TYPE ST_Zustand_Netz_Anford :
STRUCT
	Aktiv				: BOOL	;
	Temp                : REAL;
	Temp_Max            : REAL;
	Temp_Min            : REAL;
	Temp_Oben			: REAL;
	Temp_Oben_Max		: REAL	;
	Temp_Oben_Min		: REAL	;
	Temp_Unten			: REAL;
	Temp_Unten_Max		: REAL	;
	Temp_Unten_Min		: REAL	;
END_STRUCT
END_TYPE

(* stored: Version 1.1.0.1, ProductVersion 3.1.4024.10
   DUT ST_Zustand_Netz_Anford: Id {3bb66fe0-892b-4f8e-9f05-196c00cf30df} *)
